FUNCTION_BLOCK controller
  (* Standard: 61499-2 *)
  (* Version 0.1, 2017-00-25, hpea485, UOA *)
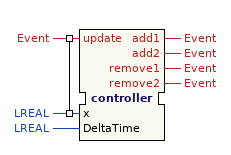
  EVENT_INPUT
    update WITH x;
  END_EVENT
  EVENT_OUTPUT
    add1;
    add2;
    remove1;
    remove2;
  END_EVENT
  VAR_INPUT
    x : LREAL;
    DeltaTime : LREAL := 0.01;
  END_VAR
  VAR
    ctime : LREAL := 0;
  END_VAR
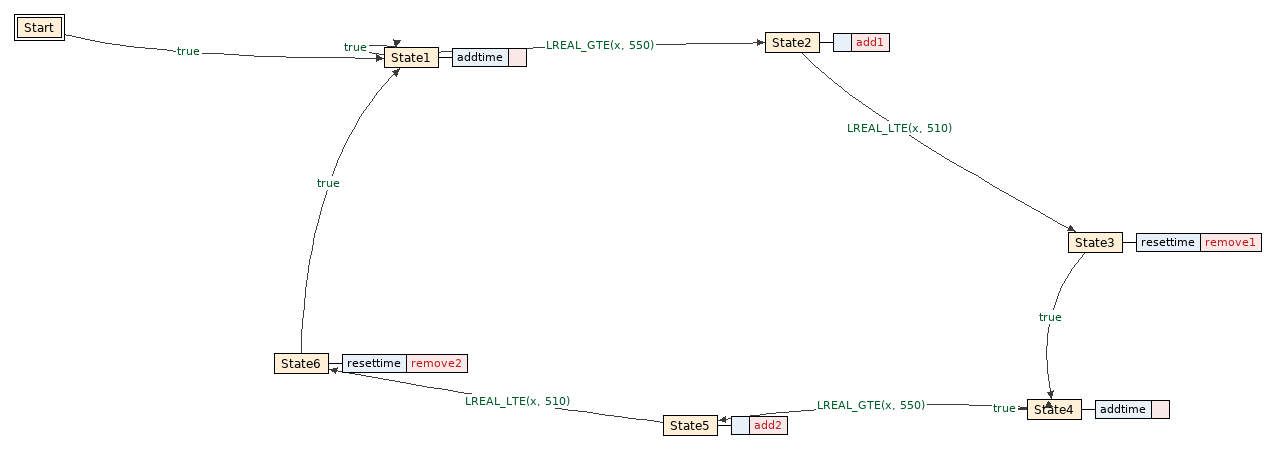
  EC_STATES
    Start;
    State1 : addtime;
    State2 : -> add1;
    State3 : resettime -> remove1;
    State4 : addtime;
    State5 : -> add2;
    State6 : resettime -> remove2;
  END_STATES
  EC_TRANSITIONS
    Start TO State1 := true;
    State1 TO State2 := LREAL_GTE(x, 550);
    State1 TO State1 := true;
    State2 TO State3 := LREAL_LTE(x, 510);
    State3 TO State4 := true;
    State4 TO State5 := LREAL_GTE(x, 550);
    State4 TO State4 := true;
    State5 TO State6 := LREAL_LTE(x, 510);
    State6 TO State1 := true;
  END_TRANSITIONS
  ALGORITHM resettime IN C:
me->ctime = 0;
  END_ALGORITHM
  ALGORITHM addtime IN C:
me->ctime += me->DeltaTime;
  END_ALGORITHM
END_FUNCTION_BLOCK
